(* CoDeSys 2.3 export: Pack9bool7SJ6xc0.EXP *)

(* POU SGL_Sismored/Sismored 4.0/Imported/Pack9bool7SJ6xc0, ST *)
FUNCTION_BLOCK Pack9bool7SJ6xc0
VAR_INPUT
	xInput1, xInput2, xInput3, xInput4, xInput5, xInput6, xInput7, xInput8, xInput9: BOOL;
END_VAR
VAR_OUTPUT
	aOutput : ARRAY[1..9] OF BOOL;
END_VAR
aOutput[1] := xInput1;
aOutput[2] := xInput2;
aOutput[3] := xInput3;
aOutput[4] := xInput4;
aOutput[5] := xInput5;
aOutput[6] := xInput6;
aOutput[7] := xInput7;
aOutput[8] := xInput8;
aOutput[9] := xInput9;

END_FUNCTION_BLOCK
